{attribute 'analysis' := '-33'}
PROGRAM INTERNAL PRG_RepeatedFieldTests
{IF defined (UNIT_TEST)}
    fbReadRepeatedFieldUint32Tests  : FB_ReadRepeatedFieldUint32Tests;
    fbReadRepeatedFieldFixed32Tests : FB_ReadRepeatedFieldFixed32Tests;
    fbReadRepeatedFieldFixed64Tests : FB_ReadRepeatedFieldFixed64Tests;
    fbReadRepeatedFieldStringTests  : FB_ReadRepeatedFieldStringTests;
    fbReadRepeatedFieldBytesTests   : FB_ReadRepeatedFieldBytesTests;
    fbReadRepeatedFieldBoolTests    : FB_ReadRepeatedFieldBoolTests;
{END_IF}

END_PROGRAM

(* stored: Version 1.1.0.1
   POU PRG_RepeatedFieldTests: Id {a1a74a7e-1fb5-4efe-992f-5a55a088b19e}, SpecialFunc None *)
